FUNCTION_BLOCK E_TP_RETRIG (* standard timer function block (pulse) - retriggerable version *)
  (* Standard: 61499-2; Classification: standard timer function block; Description: Copyright (c) 2024 HR Agrartechnik GmbH This program and the accompanying materials are made available under the terms of the Eclipse Public License 2.0 which is available at https://www.eclipse.org/legal/epl-2.0/ SPDX-License-Identifier: EPL-2.0 *)
  (* Version 1.1, 2026-04-19, Franz Höpfinger, HR Agrartechnik GmbH, retriggerable version *)
  (* Version 3.0, 2025-04-14, Patrick Aigner, changed package *)
  (* Version 1.1, 2024-04-23, Franz Hoepfinger, HR Agrartechnik GmbH, Add a Reset to Timer FBs *)
  (* Version 1.0, 2024-03-04, Franz Hoepfinger, HR Agrartechnik GmbH *)
  PACKAGE iec61499::events::timers;
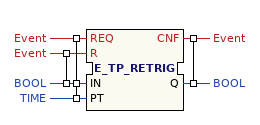
  EVENT_INPUT
    REQ WITH IN, PT; (* Service Request (Restarts the timer) *)
    R WITH IN; (* Reset *)
  END_EVENT
  EVENT_OUTPUT
    CNF WITH Q; (* Confirmation of Requested Service *)
  END_EVENT
  VAR_INPUT
    IN : BOOL; (* Input *)
    PT : TIME; (* Pulse time *)
  END_VAR
  VAR_OUTPUT
    Q : BOOL; (* Output *)
  END_VAR
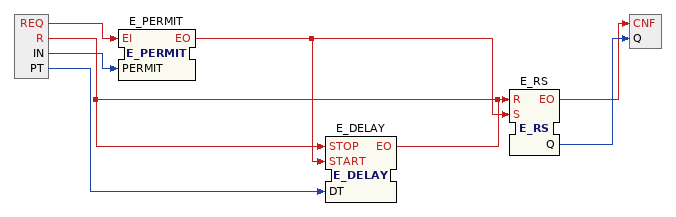
  FBS
    E_DELAY : iec61499::events::E_DELAY;
    E_RS : iec61499::events::E_RS;
    E_PERMIT : iec61499::events::E_PERMIT;
  END_FBS
  EVENT_CONNECTIONS
    E_RS.EO TO CNF;
    R TO E_DELAY.STOP;
    R TO E_RS.R;
    E_DELAY.EO TO E_RS.R;
    REQ TO E_PERMIT.EI;
    E_PERMIT.EO TO E_RS.S;
    E_PERMIT.EO TO E_DELAY.START;
  END_CONNECTIONS
  DATA_CONNECTIONS
    PT TO E_DELAY.DT;
    E_RS.Q TO Q;
    IN TO E_PERMIT.PERMIT;
  END_CONNECTIONS
END_FUNCTION_BLOCK
